{attribute 'linkalways'} 
{attribute 'no_explicit_call' := 'This FB is a CLASS and must be accessed using methods or properties'}
{attribute 'enable_dynamic_creation'}
FUNCTION_BLOCK Node_F_VN_FillContainer_REAL EXTENDS VisionNode
VAR
    ipContainer : _ITcVnContainer;
    fValue : _REAL(0);
    hrPrev : _HRESULT(S_OK);
    hresult : _HRESULT(S_OK);
END_VAR

METHOD PUBLIC  Clone : I_Node
VAR
    pNode : POINTER TO Node_F_VN_FillContainer_REAL;
END_VAR
pNode := __NEW(Node_F_VN_FillContainer_REAL);
Clone := pNode^;
END_METHOD

METHOD FB_init : BOOL
VAR_INPUT
    bInitRetains : BOOL; // if TRUE, the retain variables are initialized (warm start / cold start)
    bInCopyCode : BOOL;  // if TRUE, the instance afterwards gets moved into the copy code (online change)
END_VAR
AddInput('ipContainer', ipContainer);
AddInput('fValue', fValue);
AddInput('hrPrev', hrPrev);
AddOutput('ipContainer', ipContainer);
AddOutput('hresult',hresult);
END_METHOD

METHOD PROTECTED OnExecute : HRESULT
hresult.Value := F_VN_FillContainer_REAL(
    ipContainer := ipContainer.Value,
    fValue := fValue.Value,
    hrPrev:= hrPrev.Value);
END_METHOD

METHOD PUBLIC PreExecutionCheck
VAR_INPUT
    Check : I_PreExecutionChecks;
END_VAR
Check.IsTrue(ipContainer.IsValid, 'ipContainer must be a valid container');
END_METHOD

END_FUNCTION_BLOCK

(* stored: Version 1.1.0.1, ProductVersion 3.1.4024.13
   POU Node_F_VN_FillContainer_REAL: Id {6e92222a-25f7-4d84-9769-935b036de2de}, SpecialFunc None
   Folder Constructor: Id {e4114acd-78be-4e1b-a2e5-ae07d30dbcc0}
   Method Clone: Id {8b775a9f-3894-43d6-8832-92838eea781a}
   Method FB_init: Id {fb4574f9-c63d-41e9-a2c8-69973b2057e8}
   Method OnExecute: Id {e1a88552-b119-4dc1-9dac-58844d8c57af}
   Method PreExecutionCheck: Id {f754d8c0-6073-468d-98df-e6ab48a65da5} *)
